TYPE PowerMsg :
STRUCT
	Id : EPowerIlluminationFlow;
	Power : LREAL;
	PowerCal_mW : LREAL; 
END_STRUCT
END_TYPE

(* stored: Version 1.1.0.1, ProductVersion 3.1.4024.3
   DUT PowerMsg: Id {40dcd94b-a0db-4db3-ba5c-377bddd41d33} *)
